// TIA Portal project "OPCUA" (V16)

(* hardware
DEVICE "S71500/ET200MP station_1"  S7-1500 station
   slot 0: "Rail_0"  Rack  6ES7 590-1***0-0AA0
   slot 1: "OPCUA_Server"  CPU 1516-3 PN/DP  6ES7 516-3AN01-0AB0  V2.8
      slot 3: "CPU display_1"  6ES7591-1BA00-0AA0
      slot 32768: "PROFINET interface_1"  X1
         slot 32769: "Port_1"  X1 P1
         slot 32770: "Port_2"  X1 P2
      slot 33024: "PROFINET interface_2"  X2
         slot 33025: "Port_1"  X2 P1
      slot 33280: "DP interface_1"  X3
      slot 34817: "Virtual CP interface port_1"  Virtual CP interface port  Virtual CP interface port
*)

// ===== PLC "OPCUA_Server"  CPU 1516-3 PN/DP =====

VAR_GLOBAL   // PLC tag table "Default tag table"
   "System_Byte" AT %MB1 : Byte;
   "FirstScan" AT %M1.0 : Bool;
   "DiagStatusUpdate" AT %M1.1 : Bool;
   "AlwaysTRUE" AT %M1.2 : Bool;
   "AlwaysFALSE" AT %M1.3 : Bool;
   "Clock_Byte" AT %MB0 : Byte;
   "Clock_10Hz" AT %M0.0 : Bool;
   "Clock_5Hz" AT %M0.1 : Bool;
   "Clock_2.5Hz" AT %M0.2 : Bool;
   "Clock_2Hz" AT %M0.3 : Bool;
   "Clock_1.25Hz" AT %M0.4 : Bool;
   "Clock_1Hz" AT %M0.5 : Bool;
   "Clock_0.625Hz" AT %M0.6 : Bool;
   "Clock_0.5Hz" AT %M0.7 : Bool;
END_VAR

DATA_BLOCK "Data_DB"   // DB1
{ S7_Optimized_Access := 'TRUE' }
VERSION : 0.1
   VAR
      value : Array[0..5] of Real;
      temperature : Real := 256.8;
      "counter" : Int := 58;
      state : Bool := FALSE;
   END_VAR
BEGIN
   value[0] := 1.5;
   value[1] := 2.6;
   value[2] := 3.7;
   value[3] := 4.8;
   value[4] := 5.9;
   value[5] := 9.6;
END_DATA_BLOCK

DATA_BLOCK "Counter"   // DB2
{ S7_Optimized_Access := 'TRUE' }
VERSION : 0.1
   VAR
      iCounter : Int;
      iCounter_x1000 : Int;
      xReset_Counter : Bool;
   END_VAR
BEGIN
END_DATA_BLOCK

DATA_BLOCK "Drum_DB"   // DB4
{ S7_Optimized_Access := 'TRUE' }
VERSION : 0.1
   VAR
      rPressure : Real;
      rTemp : Real;
      rLevel : Real;
      xPump_state : Bool;
      ihours : Int;
   END_VAR
BEGIN
END_DATA_BLOCK

// folder: System blocks/Program resources

DATA_BLOCK "IEC_Counter_0_DB"   // DB3
{ S7_Optimized_Access := 'TRUE' }
AUTHOR : Simatic
FAMILY : IEC
NAME : CNTR
VERSION : 1.0
// stored: InstanceOfName IEC_COUNTER
"IEC_COUNTER"
BEGIN
END_DATA_BLOCK

// folder: (top level)

FUNCTION "FC_Counter" : Void   // FC1, LAD
{ S7_Optimized_Access := 'TRUE' }
VERSION : 0.1
   VAR_TEMP
      xResetCTU : Bool;
   END_VAR
BEGIN

REGION Network 1
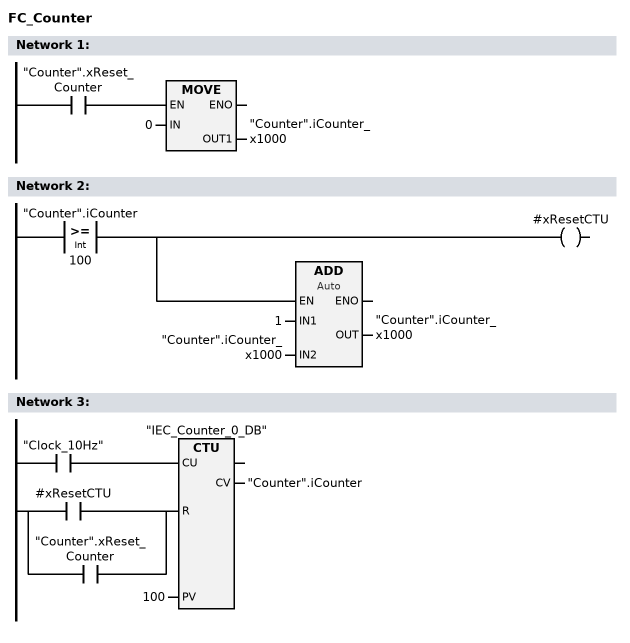
   RUNG wire#powerrail
      Contact( "Counter".xReset_Counter )
      Move(in := 0, out1 => "Counter".iCounter_x1000)
   END_RUNG
   // the same network as SCL:
   IF "Counter".xReset_Counter THEN "Counter".iCounter_x1000 := 0; END_IF;
END_REGION

REGION Network 2
   RUNG wire#powerrail
      { S7_Templates := "SrcType := Int" } GE_Contact(in1 := "Counter".iCounter, in2 := 100)
      wire#w1
      Coil( #xResetCTU )
   END_RUNG
   RUNG wire#w1
      Add(in1 := 1, in2 := "Counter".iCounter_x1000, out => "Counter".iCounter_x1000)
   END_RUNG
   // the same network as SCL:
   #xResetCTU := "Counter".iCounter >= 100;
   IF #xResetCTU THEN "Counter".iCounter_x1000 := 1 + "Counter".iCounter_x1000; END_IF;
END_REGION

REGION Network 3
   "IEC_Counter_0_DB".CTU(CU := "Clock_10Hz",
                          R := #xResetCTU OR "Counter".xReset_Counter,
                          PV := 100,
                          CV => "Counter".iCounter);
END_REGION
END_FUNCTION

ORGANIZATION_BLOCK "Main"   // OB1, LAD, ProgramCycle
TITLE = "Main Program Sweep (Cycle)"
{ S7_Optimized_Access := 'TRUE' }
VERSION : 0.1
   VAR_INPUT
      Initial_Call : Bool;   // Initial call of this OB
      Remanence : Bool;   // =True, if remanent data are available
   END_VAR
BEGIN

REGION Network 1
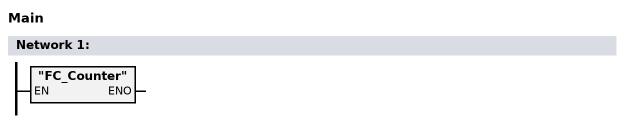
   RUNG wire#powerrail
      "FC_Counter"()
   END_RUNG
   // the same network as SCL:
   "FC_Counter"();
END_REGION
END_ORGANIZATION_BLOCK